PROGRAM MAIN
VAR
	cycler		: Cycler;
	physicalAxes: ARRAY [ShutterSide.PLUSX .. ShutterSide.MINUSX] OF AXIS_REF; (* Must be linked to Axis1 and 2, respectively, under MOTION. *)
	axisInfo	: ARRAY [ShutterSide.PLUSX..SHutterSide.MINUSX] OF AxisInfo := [(openPosition:=0.0, closedPosition:=750.0), (openPosition:=750.0, closedPosition:=0.0)];
	start, stop, reset, abort: BOOL;
	delay		: TON;
	acceleration, speed: LREAL;
	exposure	: TIME;
	

	testMotion		: TestMotion;
	home 			: BYTE;
	testMotionState	: INT :=100;
	nextInstruct	: BOOL;
END_VAR
VAR CONSTANT
	accTitle	: STRING := 'Acceleration';
END_VAR

delay(IN:=TRUE, PT:=T#0S);
IF speed>1667 THEN 
	speed:=0;
END_IF
IF delay.Q THEN
    delay(IN:=FALSE);
	
	CASE GVL.task OF
		1:
		cycler(
        	physicalAxes	:= physicalAxes,
        	axisInfo 		:= axisInfo,
        	abortRequest	:= abort,
        	resetRequest	:= reset,
        	startRequest	:= start,
        	stopRequest		:= stop,
        	exposureTime	:= exposure,
        	speed			:= speed,
        	acceleration	:= acceleration);
			
		2:
		testMotion(
			axisXP 			:= physicalAxes[ShutterSide.PLUSX],
			axisXM 			:= physicalAxes[ShutterSide.MINUSX],
			abortRequest	:= abort,
        	resetRequest	:= reset,
        	startRequest	:= start,
        	stopRequest		:= stop,
			homeRequest		:= home,
			speed			:= speed,
			state			:= testMotionState,
			nextInstruct	:= nextInstruct);

	END_CASE



END_IF

END_PROGRAM

(* stored: Version 1.1.0.1, ProductVersion 3.1.4020.12
   POU MAIN: Id {f71d400f-d229-45a7-bebf-e505112d31c1}, SpecialFunc None *)
